FUNCTION_BLOCK ServiceRegistryEntry2ServiceRegistryEntry (* Helper FB to set the connection to a Service Registry Entry type *)
  (* Standard: 61499-2; Description: Copyright (c) 2019 fortiss GmbH This program and the accompanying materials are made available under the terms of the Eclipse Public License 2.0 which is available at https://www.eclipse.org/legal/epl-2.0/ SPDX-License-Identifier: EPL-2.0 *)
  (* Version 1.0, 2019-01-28, Jose Cabral, fortiss GmbH *)
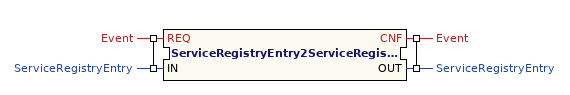
  EVENT_INPUT
    REQ WITH IN; (* Request *)
  END_EVENT
  EVENT_OUTPUT
    CNF WITH OUT; (* Confirmation *)
  END_EVENT
  VAR_INPUT
    IN : ServiceRegistryEntry; (* Input *)
  END_VAR
  VAR_OUTPUT
    OUT : ServiceRegistryEntry; (* Output *)
  END_VAR
  (* Service APPLICATION/RESOURCE: Helper FB to set the connection to a Service Registry Entry type *)
END_FUNCTION_BLOCK
